(* -----------------------------------------------------------------------------
| This sample has been supplied by Beckhoff As-Is and is intended only as an   |
| example implementation. Functionality is not guaranteed.                     |
----------------------------------------------------------------------------- *)

FUNCTION_BLOCK FB_StateMachine
VAR_INPUT
	bStart : BOOL;
	bStop : BOOL;	
	bBottle : BOOL;				// fotocellula FC1	
END_VAR
VAR_OUTPUT
	bConveyor : BOOL;			// nastro trasportatore
	bWater : BOOL;				// riempimento acqua
	bMint : BOOL;				// riempimento menta	
	bCorking : BOOL;			// inserimento del tappo
END_VAR
VAR
	nStep : INT;
	
	fbTonBottle : TON;
	fbRtBottle : R_TRIG;
	
	fbTonStep2 : TON;
	fbTonStep3 : TON;
	fbTonStep4 : TON;
	fbTonStep5 : TON;
	fbTonStep6 : TON;
END_VAR

(* -----------------------------------------------------------------------------
| This sample has been supplied by Beckhoff As-Is and is intended only as an   |
| example implementation. Functionality is not guaranteed.                     |
----------------------------------------------------------------------------- *)

(* filtri *)
fbTonBottle(IN:= bBottle, PT:= T#500MS);		// filtro sensore presenza bottiglia

(* fronti *)
fbRtBottle(CLK:= fbTonBottle.Q);

(* tempo di permanenza negli step *)
fbTonStep2(IN:= nStep = 2, PT:= T#5S);			// tempo di riempimento acqua
fbTonStep3(IN:= nStep = 3, PT:= T#1S);			// tempo di riempimento menta
fbTonStep4(IN:= nStep = 4, PT:= T#1S);			// attesa prima di tappatura
fbTonStep5(IN:= nStep = 5, PT:= T#3S);			// tempo di tappatura
fbTonStep6(IN:= nStep = 6, PT:= T#1S);			// attesa dopo tappatura

CASE nStep OF
	0: (* macchina ferma *)
		bConveyor := FALSE;
		bWater := FALSE;
		bMint := FALSE;
		bCorking := FALSE;
		
		(* transition *)
		IF NOT bStop AND bStart THEN
			nStep := 1;
		END_IF
		
	1: (* avanzamento nastro *)
		bConveyor := TRUE;
		bWater := FALSE;
		bMint := FALSE;
		bCorking := FALSE;
		
		(* transition *)
		IF fbRtBottle.Q THEN
			nStep := 2;
		END_IF
		
	2: (* riempimento acqua *)
		bConveyor := FALSE;
		bWater := TRUE;
		bMint := FALSE;
		bCorking := FALSE;
		
		(* transition *)
		IF fbTonStep2.Q THEN
			nStep := 3;
		END_IF
		
	3: (* riempimento menta *)
		bConveyor := FALSE;
		bWater := FALSE;
		bMint := TRUE;
		bCorking := FALSE;
		
		(* transition *)
		IF fbTonStep3.Q THEN
			nStep := 4;
		END_IF
		
	4: (* attesa *)
		bConveyor := FALSE;
		bWater := FALSE;
		bMint := TRUE;
		bCorking := FALSE;
		
		(* transition *)
		IF fbTonStep4.Q THEN
			nStep := 5;
		END_IF
		
	5: (* tappatura *)
		bConveyor := FALSE;
		bWater := FALSE;
		bMint := FALSE;
		bCorking := TRUE;
		
		(* transition *)
		IF fbTonStep5.Q THEN
			nStep := 6;
		END_IF
		
	6: (* attesa *)
		bConveyor := FALSE;
		bWater := FALSE;
		bMint := FALSE;
		bCorking := FALSE;
		
		(* transition *)
		IF fbTonStep6.Q THEN
			nStep := 1;
		END_IF

END_CASE

END_FUNCTION_BLOCK

(* stored: Version 1.1.0.1, ProductVersion 3.1.4024.12
   POU FB_StateMachine: Id {dc0f107e-e5d6-4626-8375-b7a8e433f6a4}, SpecialFunc None *)
